PROGRAM MAINFast
(*******************************************************************************************************
Title				:	Main program fast 
Description			:	Calling the created subroutines (Task 100µs)
Version / Date		:	1.0.0 / 23.05.2016 / created program (Version progress see below)
********************************************************************************************************)
VAR

(* Cycle counter *)
	nCycleCounter							:UDINT;
	
END_VAR
(*******************************************************************************************************
Version / Date / Description:
1.0.0   / 23.05.2016 / created program
********************************************************************************************************)
(* End *)

(* MAIN - 100µs *)

(* THIS CODE IS ONLY AN EXAMPLE - YOU HAVE TO CHECK APTITUDE FOR YOUR APPLICATION *)

(* Cycle counter *)
	nCycleCounter := nCycleCounter + 1;

	IF bMachineSequenzAktiv
	THEN
	
		(* Test Averaging *)
		AverageOut();
		
	END_IF
	
(* End *)

END_PROGRAM

(* stored: Version 1.1.0.1, ProductVersion 3.1.4020.12
   POU MAINFast: Id {9b7c0521-0ec3-464f-9e63-d2e459844049}, SpecialFunc None *)
